// TIA Portal project "mk" (V17)

(* hardware
DEVICE "S7-1500/ET200MP station_1"  S7-1500 station
   slot 0: "Rail_0"  Rack  6ES7 590-1***0-0AA0
   slot 1: "ppl"  CPU 1516-3 PN/DP  6ES7 516-3AN01-0AB0  V2.9
      slot 3: "CPU display_1"  6ES7591-1BA00-0AA0
      slot 32768: "PROFINET interface_1"  X1
         slot 32769: "Port_1"  X1 P1
         slot 32770: "Port_2"  X1 P2
      slot 33024: "PROFINET interface_2"  X2
         slot 33025: "Port_1"  X2 P1
      slot 33280: "DP interface_1"  X3
      slot 34817: "Virtual CP interface port_1"  Virtual CP interface port  Virtual CP interface port
*)

// ===== PLC "ppl"  CPU 1516-3 PN/DP =====

VAR_GLOBAL   // PLC tag table "Default tag table"
   "Tag_3" AT %Q0.0 : Bool;
   "Tag_4" AT %I0.0 : Bool;
   "Tag_5" AT %I0.1 : Bool;
   "Tag_6" AT %I0.2 : Bool;
   "Tag_7" AT %Q0.2 : Bool;
   "Tag_8" AT %I0.5 : Bool;
   "Tag_9" AT %I0.3 : Bool;
   "Tag_10" AT %QD100 : DWord;
   "Tag_11" AT %I0.4 : Bool;
   "Tag_12" AT %Q0.1 : Bool;
   "Tag_13" AT %ID100 : DWord;
   "Tag_14" AT %QD0 : Real;
   "Tag_15" AT %QD4 : DWord;
   "Tag_1" AT %IW64 : Word;
   "Tag_2" AT %MD0 : Real;
   "Tag_16" AT %QW64 : Int;
   "Tag_17" AT %M0.0 : Bool;
   "Tag_18" AT %M0.1 : Bool;
   "Tag_19" AT %M0.4 : Bool;
   "Tag_20" AT %M0.5 : Bool;
   "Tag_21" AT %M0.6 : Bool;
   "Tag_22" AT %M0.7 : Bool;
END_VAR

// folder: System blocks/Program resources

DATA_BLOCK "IEC_Counter_0_DB"   // DB1
{ S7_Optimized_Access := 'FALSE' }
AUTHOR : Simatic
FAMILY : IEC
NAME : CNTR
VERSION : 1.0
// stored: InstanceOfName IEC_COUNTER
"IEC_COUNTER"
BEGIN
END_DATA_BLOCK

DATA_BLOCK "IEC_Timer_0_DB"   // DB2
{ S7_Optimized_Access := 'FALSE' }
AUTHOR : Simatic
FAMILY : IEC
NAME : IEC_TMR
VERSION : 1.0
// stored: InstanceOfName IEC_TIMER
"IEC_TIMER"
BEGIN
END_DATA_BLOCK

DATA_BLOCK "IEC_Timer_0_DB_1"   // DB3
{ S7_Optimized_Access := 'FALSE' }
AUTHOR : Simatic
FAMILY : IEC
NAME : IEC_TMR
VERSION : 1.0
// stored: InstanceOfName IEC_TIMER
"IEC_TIMER"
BEGIN
END_DATA_BLOCK

DATA_BLOCK "IEC_Timer_0_DB_2"   // DB4
{ S7_Optimized_Access := 'TRUE' }
AUTHOR : Simatic
FAMILY : IEC
NAME : IEC_TMR
VERSION : 1.0
// stored: InstanceOfName IEC_TIMER
"IEC_TIMER"
BEGIN
END_DATA_BLOCK

// folder: (top level)

ORGANIZATION_BLOCK "Main"   // OB1, LAD, ProgramCycle
TITLE = "Main Program Sweep (Cycle)"
{ S7_Optimized_Access := 'TRUE' }
VERSION : 0.1
   VAR_INPUT
      Initial_Call : Bool;   // Initial call of this OB
      Remanence : Bool;   // =True, if remanent data are available
   END_VAR
BEGIN

REGION Network 1: Control Panel
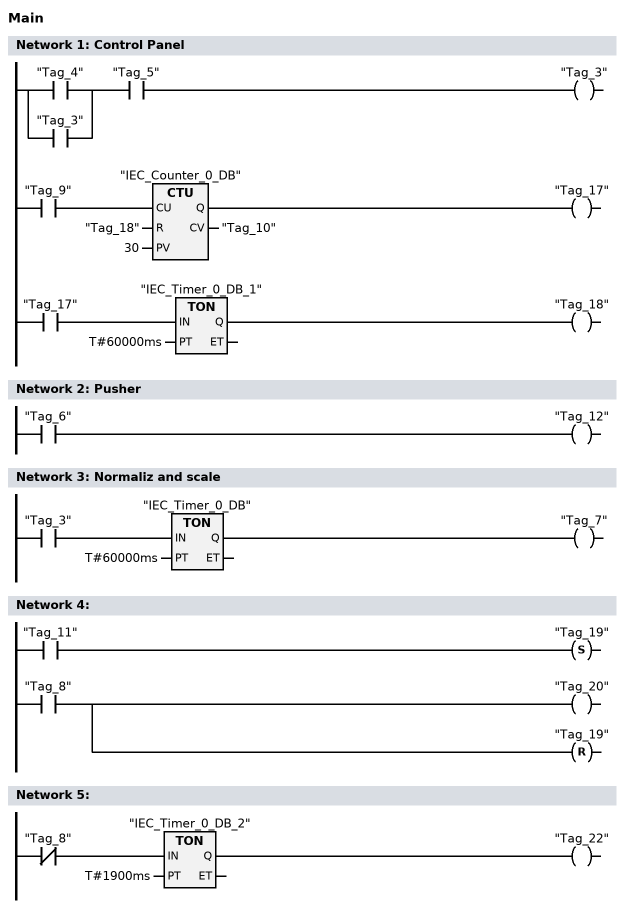
   "Tag_3" := ("Tag_4" OR "Tag_3") AND "Tag_5";
   "IEC_Counter_0_DB".CTU(CU := "Tag_9", R := "Tag_18", PV := 30, CV => "Tag_10");
   "Tag_17" := "IEC_Counter_0_DB".Q;
   "IEC_Timer_0_DB_1".TON(IN := "Tag_17", PT := T#60000ms);
   "Tag_18" := "IEC_Timer_0_DB_1".Q;
END_REGION

REGION Network 2: Pusher
   RUNG wire#powerrail
      Contact( "Tag_6" )
      Coil( "Tag_12" )
   END_RUNG
   // the same network as SCL:
   "Tag_12" := "Tag_6";
END_REGION

REGION Network 3: Normaliz and scale
   "IEC_Timer_0_DB".TON(IN := "Tag_3", PT := T#60000ms);
   "Tag_7" := "IEC_Timer_0_DB".Q;
END_REGION

REGION Network 4
   RUNG wire#powerrail
      Contact( "Tag_11" )
      S_Coil( "Tag_19" )
   END_RUNG
   RUNG wire#powerrail
      Contact( "Tag_8" )
      wire#w1
      Coil( "Tag_20" )
   END_RUNG
   RUNG wire#w1
      R_Coil( "Tag_19" )
   END_RUNG
   // the same network as SCL:
   IF "Tag_11" THEN "Tag_19" := TRUE; END_IF;
   "Tag_20" := "Tag_8";
   IF "Tag_8" THEN "Tag_19" := FALSE; END_IF;
END_REGION

REGION Network 5
   "IEC_Timer_0_DB_2".TON(IN := NOT "Tag_8", PT := T#1900ms);
   "Tag_22" := "IEC_Timer_0_DB_2".Q;
END_REGION
END_ORGANIZATION_BLOCK